// TIA Portal project "Manual RoboCrane full program" (V16)

(* hardware
DEVICE "S71500/ET200MP station_1"  S7-1500 station
   slot 0: "Rail_0"  Rack  6ES7 590-1***0-0AA0
   slot 1: "PLC_1"  CPU 1516F-3 PN/DP  6ES7 516-3FN01-0AB0  V1.8
      slot 3: "CPU display_1"  6ES7591-1BA00-0AA0
      slot 32768: "PROFINET interface_1"  X1
         slot 32769: "Port_1"  X1 P1
         slot 32770: "Port_2"  X1 P2
      slot 33024: "PROFINET interface_2"  X2
         slot 33025: "Port_1"  X2 P1
      slot 33280: "DP interface_1"  X3
   slot 2: "DI 32x24VDC HF_1"  DI 32x24VDC HF  6ES7 521-1BL00-0AB0  V2.1
   slot 3: "DQ 32x24VDC/0.5A ST_1"  DQ 32x24VDC/0.5A ST  6ES7 522-1BL00-0AB0  V2.0
   slot 4: "AI 8xU/I/RTD/TC ST_1"  AI 8xU/I/RTD/TC ST  6ES7 531-7KF00-0AB0  V2.0
   slot 5: "AQ 4xU/I ST_1"  AQ 4xU/I ST  6ES7 532-5HD00-0AB0  V2.0
*)

// ===== PLC "PLC_1"  CPU 1516F-3 PN/DP =====

VAR_GLOBAL   // PLC tag table "OPTS_tag_table"
   "ButtonFirstJointUp" AT %I2.4 : Bool;
   "FL_PositionSensor" AT %IW126 : Int;
   "FR_PositionSensor" AT %IW128 : Int;
   "FirstJoint_PositionSensor" AT %IW130 : Int;
   "SensorXValue" AT %IW132 : Int;
   "SensorYValue" AT %IW134 : Int;
   "BaseUp" AT %QW4 : Word;
   "ButtonBaseLeft" AT %I2.2 : Bool;
   "ButtonBaseRight" AT %I2.3 : Bool;
   "ButtonBaseUp" AT %I2.0 : Bool;
   "ButtonBaseDown" AT %I2.1 : Bool;
   "BaseLeft" AT %QW6 : Word;
   "ButtonFirstJointDown" AT %I2.5 : Bool;
   "FirstJointUp" AT %Q10.0 : Bool;
   "FirstJointDown" AT %Q10.1 : Bool;
   "StepperRotCW" AT %Q10.2 : Bool;
   "StepperRotCCW" AT %Q10.3 : Bool;
   "StepperTelescoCW" AT %Q10.4 : Bool;
   "StepperTelescoCCW" AT %Q10.5 : Bool;
   "ServoCW" AT %Q10.6 : Bool;
   "ServoCCW" AT %Q10.7 : Bool;
   "ButtonSecondJointUp" AT %I2.6 : Bool;
   "ButtonSecondJointDown" AT %I2.7 : Bool;
   "ButtonThirdJointUp" AT %I3.0 : Bool;
   "ButtonFourthJointUp" AT %I3.2 : Bool;
   "ButtonFourthJointDown" AT %I3.3 : Bool;
   "ButtonStepperRotCW" AT %I3.4 : Bool;
   "ButtonThirdJointDown" AT %I3.1 : Bool;
   "ButtonStepperRotCCW" AT %I3.5 : Bool;
   "ButtonServoCW" AT %I3.6 : Bool;
   "ButtonServoCCW" AT %I3.7 : Bool;
   "SecondJoint_PositionSensor" AT %IW136 : Int;
   "ThirdJoint_PositionSensor" AT %IW138 : Int;
   "FourthJoint_PositionSensor" AT %IW140 : Int;
   "SecondJoint" AT %QW0 : Word;
   "ThirdJoint" AT %QW2 : Word;
   "FourthJointUp" AT %Q11.0 : Bool;
   "FourthJointDown" AT %Q11.1 : Bool;
END_VAR

DATA_BLOCK "Base Movement Buttons_DB"   // DB1
{ S7_Optimized_Access := 'TRUE' }
VERSION : 0.1
// stored: InstanceOfName Base Movement Buttons
"Base Movement Buttons"
BEGIN
END_DATA_BLOCK

DATA_BLOCK "movement analog_DB"   // DB2
{ S7_Optimized_Access := 'TRUE' }
VERSION : 0.1
// stored: InstanceOfName movement analog
"movement analog"
BEGIN
END_DATA_BLOCK

DATA_BLOCK "motor_position_DB"   // DB3
{ S7_Optimized_Access := 'TRUE' }
VERSION : 0.1
// stored: InstanceOfName motor_position
"motor_position"
BEGIN
END_DATA_BLOCK

DATA_BLOCK "movement analog_DB_1"   // DB4
{ S7_Optimized_Access := 'TRUE' }
VERSION : 0.1
// stored: InstanceOfName movement analog
"movement analog"
BEGIN
END_DATA_BLOCK

DATA_BLOCK "movement digital_DB"   // DB5
{ S7_Optimized_Access := 'TRUE' }
VERSION : 0.1
// stored: InstanceOfName movement digital
"movement digital"
BEGIN
END_DATA_BLOCK

DATA_BLOCK "movement analog_DB_2"   // DB6
{ S7_Optimized_Access := 'TRUE' }
VERSION : 0.1
// stored: InstanceOfName movement analog
"movement analog"
BEGIN
END_DATA_BLOCK

DATA_BLOCK "movement analog_DB_3"   // DB7
{ S7_Optimized_Access := 'TRUE' }
VERSION : 0.1
// stored: InstanceOfName movement analog
"movement analog"
BEGIN
END_DATA_BLOCK

DATA_BLOCK "movement analog_DB_4"   // DB9
{ S7_Optimized_Access := 'TRUE' }
VERSION : 0.1
// stored: InstanceOfName movement analog
"movement analog"
BEGIN
END_DATA_BLOCK

DATA_BLOCK "movement digital_DB_telescop"   // DB10
{ S7_Optimized_Access := 'TRUE' }
VERSION : 0.1
// stored: InstanceOfName movement digital
"movement digital"
BEGIN
END_DATA_BLOCK

DATA_BLOCK "movement digital_DB_rotate_base"   // DB11
{ S7_Optimized_Access := 'TRUE' }
VERSION : 0.1
// stored: InstanceOfName movement digital
"movement digital"
BEGIN
END_DATA_BLOCK

DATA_BLOCK "movement digital_DB-Servo"   // DB12
{ S7_Optimized_Access := 'TRUE' }
VERSION : 0.1
// stored: InstanceOfName movement digital
"movement digital"
BEGIN
END_DATA_BLOCK

DATA_BLOCK "movement digital_DBFourthJoint"   // DB14
{ S7_Optimized_Access := 'TRUE' }
VERSION : 0.1
// stored: InstanceOfName movement digital
"movement digital"
BEGIN
END_DATA_BLOCK

FUNCTION_BLOCK "Base Movement Buttons"   // FB1, FBD
{ S7_Optimized_Access := 'TRUE' }
VERSION : 0.1
// !!You stand in front of the OPTS, the two motors in the front are the ones we talk about while programming. This means that 'Up' is the left front motor going up. 'Left' is the front right motor going up.
   VAR_INPUT
      buttonBaseUp : Bool;
      buttonBaseDown : Bool;
      buttonBaseLeft : Bool;
      buttonBaseRight : Bool;
      doNotMoveFrontLeftUp : Bool;
      doNotMoveFrontLeftDown : Bool;
      doNotMoveFrontRightUp : Bool;
      doNotMoveFrontRightDown : Bool;
      doNotMoveFirstJointUp : Bool;
      doNotMoveFirstJointDown : Bool;
      buttonFirstJointUp : Bool;
      buttonFirstJointDown : Bool;
   END_VAR
   VAR_OUTPUT
      baseUp : Word;
      baseLeft : Word;
      firstJointUp : Bool;
      firstJointDown : Bool;
   END_VAR
   VAR
      pTrigDown : Bool;
      pTrigUp : Bool;
      pTrigLeft : Bool;
      pTrigRight : Bool;
   END_VAR
   VAR_TEMP   // added for the SCL form of the ladder/FBD networks
      _w1 : Bool;
      _w2 : Bool;
   END_VAR
BEGIN

REGION Network 1
   // Base Up(Analog)
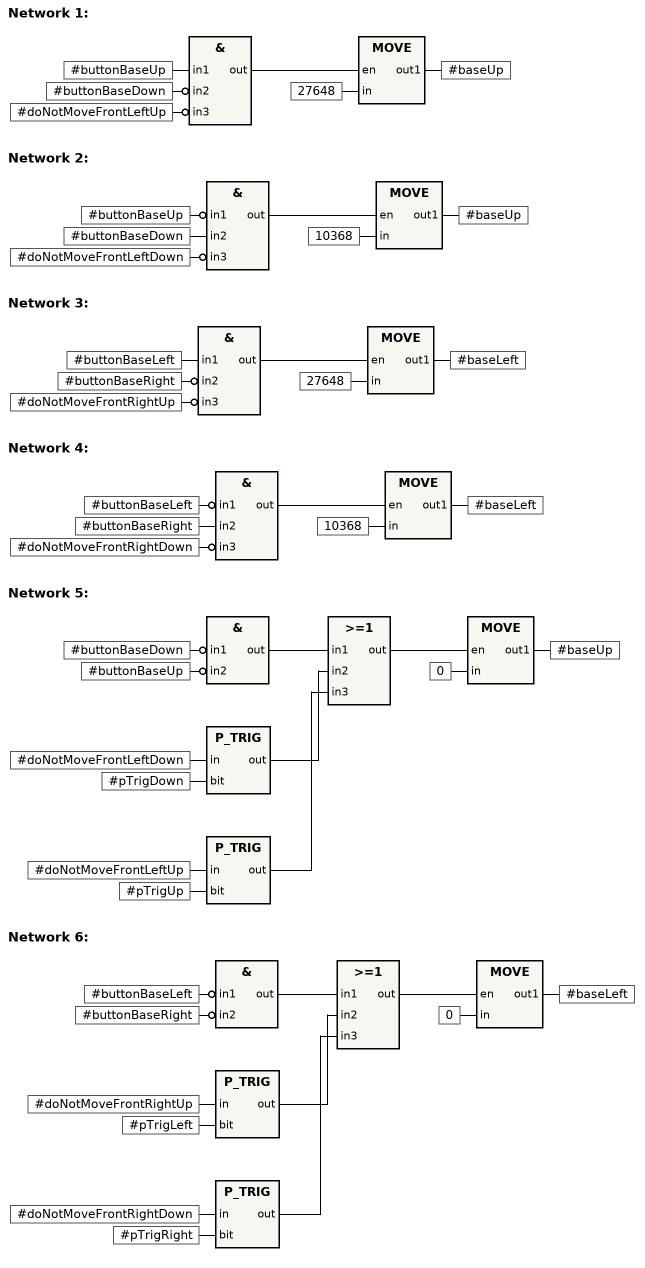
   IF #buttonBaseUp AND NOT #buttonBaseDown AND NOT #doNotMoveFrontLeftUp THEN #baseUp := 27648; END_IF;
END_REGION

REGION Network 2
   // Base Down(Analog)
   IF NOT #buttonBaseUp AND #buttonBaseDown AND NOT #doNotMoveFrontLeftDown THEN #baseUp := 10368; END_IF;
END_REGION

REGION Network 3
   // Base Left(Analog)
   IF #buttonBaseLeft AND NOT #buttonBaseRight AND NOT #doNotMoveFrontRightUp THEN
       #baseLeft := 27648;
   END_IF;
END_REGION

REGION Network 4
   // Base Right(Analog)
   IF NOT #buttonBaseLeft AND #buttonBaseRight AND NOT #doNotMoveFrontRightDown THEN
       #baseLeft := 10368;
   END_IF;
END_REGION

REGION Network 5
   // If there is no button pressed, the motors won't move.
   #_w1 := #doNotMoveFrontLeftDown AND NOT #pTrigDown;   // rising edge
   #pTrigDown := #doNotMoveFrontLeftDown;
   #_w2 := #doNotMoveFrontLeftUp AND NOT #pTrigUp;   // rising edge
   #pTrigUp := #doNotMoveFrontLeftUp;
   IF (NOT #buttonBaseDown AND NOT #buttonBaseUp) OR #_w1 OR #_w2 THEN #baseUp := 0; END_IF;
END_REGION

REGION Network 6
   // Same as Network 5, but with Left and Right.
   #_w1 := #doNotMoveFrontRightUp AND NOT #pTrigLeft;   // rising edge
   #pTrigLeft := #doNotMoveFrontRightUp;
   #_w2 := #doNotMoveFrontRightDown AND NOT #pTrigRight;   // rising edge
   #pTrigRight := #doNotMoveFrontRightDown;
   IF (NOT #buttonBaseLeft AND NOT #buttonBaseRight) OR #_w1 OR #_w2 THEN #baseLeft := 0; END_IF;
END_REGION

REGION Network 7
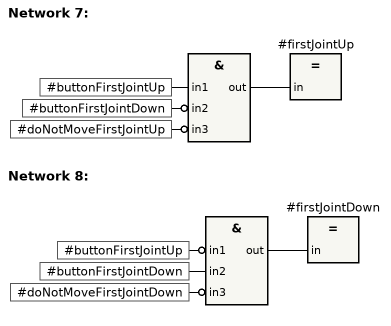
   #firstJointUp := #buttonFirstJointUp AND NOT #buttonFirstJointDown AND NOT #doNotMoveFirstJointUp;
END_REGION

REGION Network 8
   #firstJointDown := NOT #buttonFirstJointUp AND #buttonFirstJointDown AND NOT #doNotMoveFirstJointDown;
END_REGION
END_FUNCTION_BLOCK

FUNCTION_BLOCK "motor_position"   // FB2, FBD
{ S7_Optimized_Access := 'TRUE' }
VERSION : 0.1
   VAR_INPUT
      frontLeft : Int;
      frontRight : Int;
      firstJoint : Int;
      secondJoint : Int;
      thirdJoint : Int;
      fouthJoint : Int;
   END_VAR
   VAR_OUTPUT
      limitTopLeft : Bool;
      limitBottomLeft : Bool;
      limitTopRight : Bool;
      limitBottomRight : Bool;
      limitJoint_1_Top : Bool;
      limitJoint_1_Bottom : Bool;
      limitJoint_2_Top : Bool := false;
      limitJoint_2_Bottom : Bool := false;
      limitJoint_3_Top : Bool := false;
      limitJoint_3_Bottom : Bool := false;
      limitJoint_4_Top : Bool := false;
      limitJoint_4_Bottom : Bool := false;
   END_VAR
BEGIN

REGION Network 1
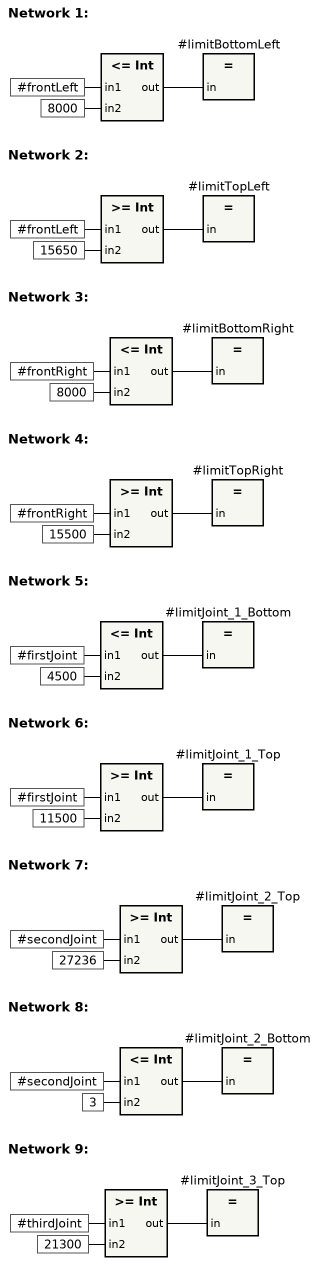
   #limitBottomLeft := #frontLeft <= 8000;
END_REGION

REGION Network 2
   #limitTopLeft := #frontLeft >= 15650;
END_REGION

REGION Network 3
   #limitBottomRight := #frontRight <= 8000;
END_REGION

REGION Network 4
   #limitTopRight := #frontRight >= 15500;
END_REGION

REGION Network 5
   #limitJoint_1_Bottom := #firstJoint <= 4500;
END_REGION

REGION Network 6
   #limitJoint_1_Top := #firstJoint >= 11500;
END_REGION

REGION Network 7
   // to do
   #limitJoint_2_Top := #secondJoint >= 27236;
END_REGION

REGION Network 8
   // to do
   #limitJoint_2_Bottom := #secondJoint <= 3;
END_REGION

REGION Network 9
   // to do
   #limitJoint_3_Top := #thirdJoint >= 21300;
END_REGION

REGION Network 10
   // to do
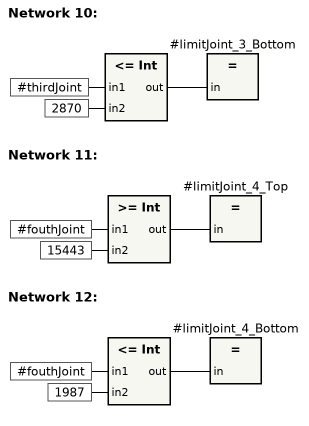
   #limitJoint_3_Bottom := #thirdJoint <= 2870;
END_REGION

REGION Network 11
   // to do
   #limitJoint_4_Top := #fouthJoint >= 15443;
END_REGION

REGION Network 12
   // to do
   #limitJoint_4_Bottom := #fouthJoint <= 1987;
END_REGION
END_FUNCTION_BLOCK

FUNCTION_BLOCK "Gyroscopic Data"   // FB3, FBD
{ S7_Optimized_Access := 'TRUE' }
VERSION : 0.1
   VAR_INPUT
      sensorXValue : Int;
      sensorYValue : Int;
   END_VAR
   VAR_OUTPUT
      stableXValue : Int;
      stableYValue : Int;
   END_VAR
BEGIN
END_FUNCTION_BLOCK

FUNCTION_BLOCK "movement analog"   // FB4, FBD
{ S7_Optimized_Access := 'TRUE' }
VERSION : 0.1
   VAR_INPUT
      up : Bool;
      down : Bool;
      limitTop : Bool;
      limitBottom : Bool;
   END_VAR
   VAR_OUTPUT
      moveBase : Word;
   END_VAR
   VAR
      pTrigDown : Bool := false;
      pTrigUp : Bool := false;
   END_VAR
   VAR_TEMP   // added for the SCL form of the ladder/FBD networks
      _w1 : Bool;
      _w2 : Bool;
   END_VAR
BEGIN

REGION Network 1
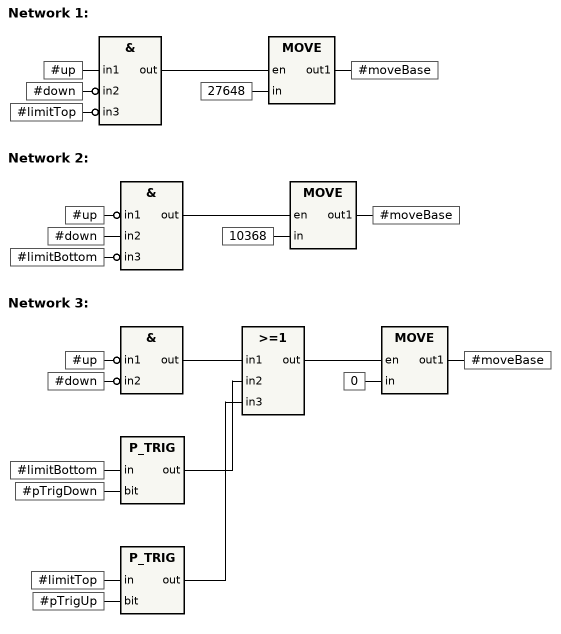
   IF #up AND NOT #down AND NOT #limitTop THEN #moveBase := 27648; END_IF;
END_REGION

REGION Network 2
   IF NOT #up AND #down AND NOT #limitBottom THEN #moveBase := 10368; END_IF;
END_REGION

REGION Network 3
   #_w1 := #limitBottom AND NOT #pTrigDown;   // rising edge
   #pTrigDown := #limitBottom;
   #_w2 := #limitTop AND NOT #pTrigUp;   // rising edge
   #pTrigUp := #limitTop;
   IF (NOT #up AND NOT #down) OR #_w1 OR #_w2 THEN #moveBase := 0; END_IF;
END_REGION
END_FUNCTION_BLOCK

FUNCTION_BLOCK "movement digital"   // FB5, FBD
{ S7_Optimized_Access := 'TRUE' }
VERSION : 0.1
   VAR_INPUT
      up : Bool;
      down : Bool;
      limitTop : Bool;
      limitBottom : Bool;
   END_VAR
   VAR_OUTPUT
      moveUp : Bool;
      moveDown : Bool;
   END_VAR
BEGIN

REGION Network 1
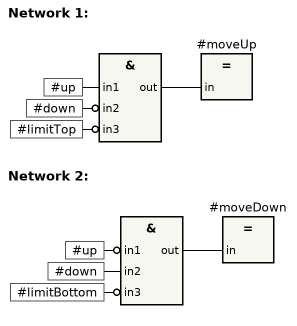
   #moveUp := #up AND NOT #down AND NOT #limitTop;
END_REGION

REGION Network 2
   #moveDown := NOT #up AND #down AND NOT #limitBottom;
END_REGION
END_FUNCTION_BLOCK

FUNCTION "movement" : Void   // FC1, FBD
{ S7_Optimized_Access := 'TRUE' }
VERSION : 0.1
   VAR_INPUT
      buttonBaseUp : Bool;   // false
      buttonBaseDown : Bool;   // false
      buttonBaseLeft : Bool;   // false
      buttonBaseRight : Bool;   // false
      buttonFirstJointUp : Bool;   // false
      buttonFirstJointDown : Bool;   // false
      buttonSecondJointUp : Bool;
      buttonSecondJointDown : Bool;
      buttonThirdJointUp : Bool;
      buttonThirdJointDown : Bool;
      buttonFourthJointUp : Bool;
      buttonFourthJointDown : Bool;
      buttonFiftJointLeft : Bool;
      buttonFiftJointRight : Bool;
      buttonRotateLeft : Bool;
      buttonRotateRight : Bool;
   END_VAR
   VAR_OUTPUT
      BaseFrontLeft : Word;
      BaseFrontRight : Word;
      firstJointUp : Bool;   // false
      firstJointDown : Bool;   // false
      secondJoint : Word;
      thirdJoint : Word;
      fourthJointUp : Bool;
      fourthJointDown : Bool;
      fiftJointUp : Bool;
      fiftJointDown : Bool;
      rotateLeft : Bool;
      rotateRight : Bool;
   END_VAR
BEGIN

REGION Network 1
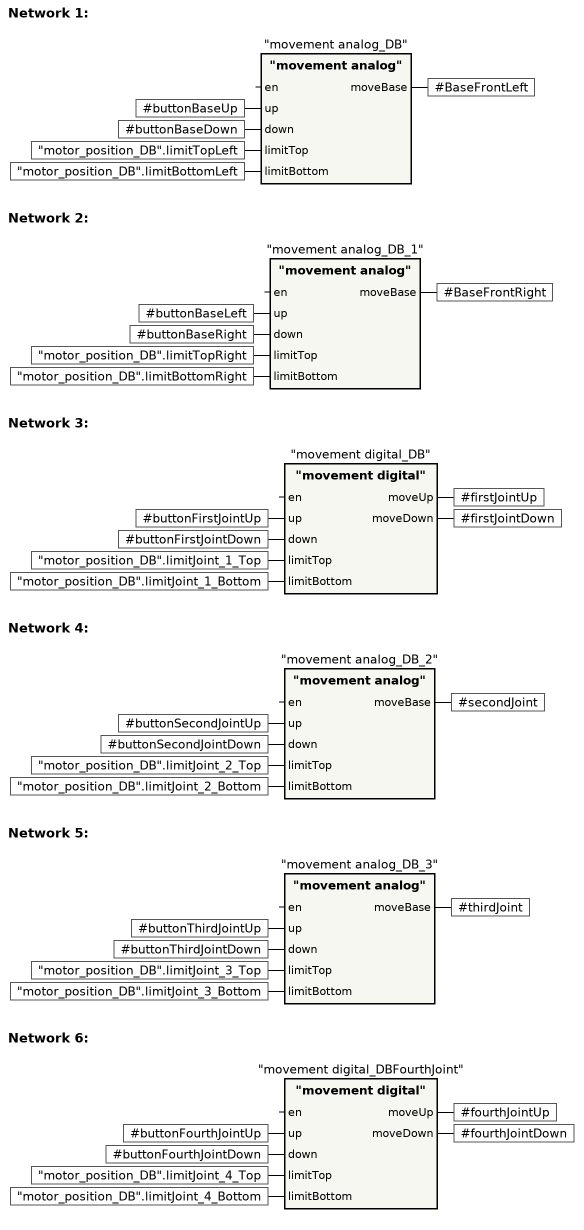
   "movement analog_DB"(up := #buttonBaseUp,   // "movement analog"
                        down := #buttonBaseDown,
                        limitTop := "motor_position_DB".limitTopLeft,
                        limitBottom := "motor_position_DB".limitBottomLeft,
                        moveBase => #BaseFrontLeft);
END_REGION

REGION Network 2
   "movement analog_DB_1"(up := #buttonBaseLeft,   // "movement analog"
                          down := #buttonBaseRight,
                          limitTop := "motor_position_DB".limitTopRight,
                          limitBottom := "motor_position_DB".limitBottomRight,
                          moveBase => #BaseFrontRight);
END_REGION

REGION Network 3
   // first joint
   "movement digital_DB"(up := #buttonFirstJointUp,   // "movement digital"
                         down := #buttonFirstJointDown,
                         limitTop := "motor_position_DB".limitJoint_1_Top,
                         limitBottom := "motor_position_DB".limitJoint_1_Bottom,
                         moveUp => #firstJointUp,
                         moveDown => #firstJointDown);
END_REGION

REGION Network 4
   // second joint
   "movement analog_DB_2"(up := #buttonSecondJointUp,   // "movement analog"
                          down := #buttonSecondJointDown,
                          limitTop := "motor_position_DB".limitJoint_2_Top,
                          limitBottom := "motor_position_DB".limitJoint_2_Bottom,
                          moveBase => #secondJoint);
END_REGION

REGION Network 5
   // third joint
   "movement analog_DB_3"(up := #buttonThirdJointUp,   // "movement analog"
                          down := #buttonThirdJointDown,
                          limitTop := "motor_position_DB".limitJoint_3_Top,
                          limitBottom := "motor_position_DB".limitJoint_3_Bottom,
                          moveBase => #thirdJoint);
END_REGION

REGION Network 6
   // fourth joint
   "movement digital_DBFourthJoint"(up := #buttonFourthJointUp,   // "movement digital"
                           down := #buttonFourthJointDown,
                           limitTop := "motor_position_DB".limitJoint_4_Top,
                           limitBottom := "motor_position_DB".limitJoint_4_Bottom,
                           moveUp => #fourthJointUp,
                           moveDown => #fourthJointDown);
END_REGION

REGION Network 7
   // fIFT JOINT (SERVO)
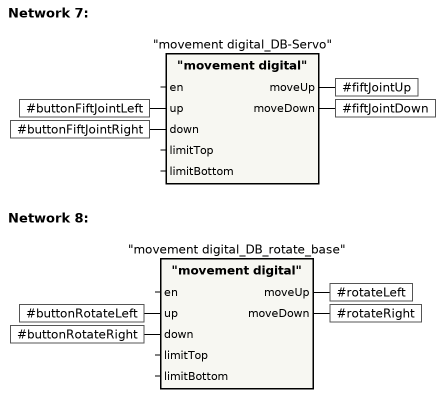
   "movement digital_DB-Servo"(up := #buttonFiftJointLeft,   // "movement digital"
                           down := #buttonFiftJointRight,
                           moveUp => #fiftJointUp,
                           moveDown => #fiftJointDown);
END_REGION

REGION Network 8
   "movement digital_DB_rotate_base"(up := #buttonRotateLeft,   // "movement digital"
                           down := #buttonRotateRight,
                           moveUp => #rotateLeft,
                           moveDown => #rotateRight);
END_REGION
END_FUNCTION

ORGANIZATION_BLOCK "Main"   // OB1, FBD, ProgramCycle
TITLE = "Main Program Sweep (Cycle)"
{ S7_Optimized_Access := 'TRUE' }
VERSION : 0.1
   VAR_INPUT
      Initial_Call : Bool;   // Initial call of this OB
      Remanence : Bool;   // =True, if remanent data are available
   END_VAR
   VAR_TEMP
      flInTemp : Real;
      frInTemp : Real;
      blInTemp : Real;
      brInTemp : Real;
   END_VAR
BEGIN

REGION Network 1
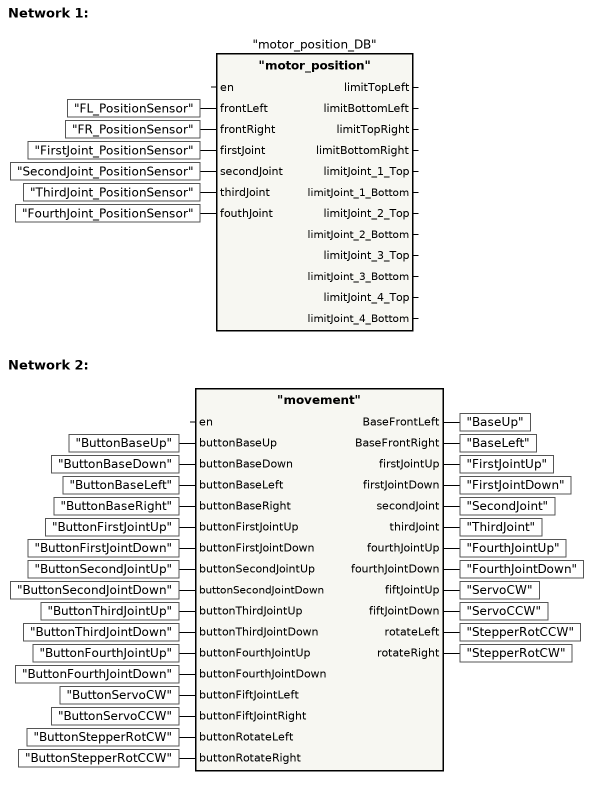
   "motor_position_DB"(frontLeft := "FL_PositionSensor",   // "motor_position"
                       frontRight := "FR_PositionSensor",
                       firstJoint := "FirstJoint_PositionSensor",
                       secondJoint := "SecondJoint_PositionSensor",
                       thirdJoint := "ThirdJoint_PositionSensor",
                       fouthJoint := "FourthJoint_PositionSensor");
END_REGION

REGION Network 2
   "movement"(buttonBaseUp := "ButtonBaseUp",
              buttonBaseDown := "ButtonBaseDown",
              buttonBaseLeft := "ButtonBaseLeft",
              buttonBaseRight := "ButtonBaseRight",
              buttonFirstJointUp := "ButtonFirstJointUp",
              buttonFirstJointDown := "ButtonFirstJointDown",
              buttonSecondJointUp := "ButtonSecondJointUp",
              buttonSecondJointDown := "ButtonSecondJointDown",
              buttonThirdJointUp := "ButtonThirdJointUp",
              buttonThirdJointDown := "ButtonThirdJointDown",
              buttonFourthJointUp := "ButtonFourthJointUp",
              buttonFourthJointDown := "ButtonFourthJointDown",
              buttonFiftJointLeft := "ButtonServoCW",
              buttonFiftJointRight := "ButtonServoCCW",
              buttonRotateLeft := "ButtonStepperRotCW",
              buttonRotateRight := "ButtonStepperRotCCW",
              BaseFrontLeft => "BaseUp",
              BaseFrontRight => "BaseLeft",
              firstJointUp => "FirstJointUp",
              firstJointDown => "FirstJointDown",
              secondJoint => "SecondJoint",
              thirdJoint => "ThirdJoint",
              fourthJointUp => "FourthJointUp",
              fourthJointDown => "FourthJointDown",
              fiftJointUp => "ServoCW",
              fiftJointDown => "ServoCCW",
              rotateLeft => "StepperRotCCW",
              rotateRight => "StepperRotCW");
END_REGION
END_ORGANIZATION_BLOCK